FUNCTION_BLOCK Drill (* Drill *)
  (* Standard: 61499-2 *)
  (* Version 0.2, 2003-12-04, JHC, Rockwell Automation, Renamed for better indexing. *)
  (* Version 0.1, 2002-11-05, JHC, Rockwell Automation, Corrected missing ST element in Algorithm REQ. *)
  (* Version 0.0, 2000-05-30, JHC, Rockwell Automation *)
  (* Compiler header: package fb.rt.benchmarks.DrillStation; *)
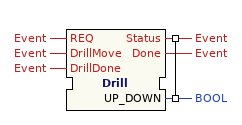
  EVENT_INPUT
    REQ; (* Normal Execution Request *)
    DrillMove; (* Simulate the time taken to move the drill *)
    DrillDone; (* Simulate the time taken to drill *)
  END_EVENT
  EVENT_OUTPUT
    Status WITH UP_DOWN;
    Done; (* Done drilling *)
  END_EVENT
  VAR_OUTPUT
    UP_DOWN : BOOL := true; (* true: up, false: down *)
  END_VAR
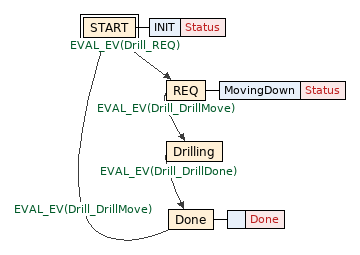
  EC_STATES
    START : INIT -> Status; (* Initial State *)
    REQ : MovingDown -> Status; (* Normal execution *)
    Done : -> Done;
    Drilling;
  END_STATES
  EC_TRANSITIONS
    START TO REQ := EVAL_EV(Drill_REQ);
    Done TO START := EVAL_EV(Drill_DrillMove);
    REQ TO Drilling := EVAL_EV(Drill_DrillMove);
    Drilling TO Done := EVAL_EV(Drill_DrillDone);
  END_TRANSITIONS
  ALGORITHM INIT IN ST: (* Initialization algorithm *)
VAL_OF_UP_DOWN()= 1;
  END_ALGORITHM
  ALGORITHM MovingDown IN ST: (* Normally executed algorithm *)
VAL_OF_UP_DOWN()= 0;
  END_ALGORITHM
END_FUNCTION_BLOCK
